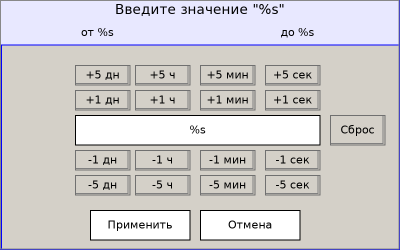
VISUALIZATION TimeInput  // 400x250
VAR_INPUT
	stVariableValue : STRING;
	stMin : STRING;
	stMax : STRING;
	wstTitle : WSTRING;
	flags : DWORD;
END_VAR
VAR
	bInit 			: BOOL;
	stMessage 		: STRING;
	stOutputValue 	: STRING;
	iCaretPosition	: INT;
	iSelectionStart	: INT;
	iSelectionEnd	: INT;
	xAllSelected	: BOOL;
END_VAR
    Rectangle (0,0 400x250)
    Rectangle (200,210 100x30), "Отмена"
        OnMouseDown: CloseDialog Dialog=TimeInput, Result=Cancel, NumpadKeypadSet=True
    Rectangle (90,210 100x30), "Применить"
        OnMouseUp: CloseDialog Dialog=TimeInput, Result=Yes, NumpadKeypad=True, NumpadKeypadSet=True
    Rectangle (0,0 400x45), "Введите значение "%s"", text variable: Header
    Button (265,90 55x20), "+1 сек", invisible if: (MinTime + T#1s >= MaxTime)
        OnMouseUp: execute {
            IF ((timevar+T#1S <= MaxTime ) AND
            			(timevar+T#1S > TimeVar)) THEN
            	timevar:=timevar+T#1S;
            END_IF
        }
    Rectangle (75,115 245x30), "%s", text variable: TIME_TO_WSTRING_HMI(TimeVar)
        p4168582468: "Время"
    Button (265,65 55x20), "+5 сек", invisible if: (MinTime + T#5s >= MaxTime)
        OnMouseUp: execute {
            IF ((timevar+T#5S <= MaxTime ) AND
            			(timevar+T#5S > TimeVar)) THEN
            	timevar:=timevar+T#5S;
            ELSE
            	timevar:=MaxTime;
            END_IF
        }
    Button (265,175 55x20), "-5 сек", invisible if: (MinTime + T#5s) >= MaxTime
        OnMouseUp: execute {
            IF (((timevar-T#5S) >= MinTime)AND
            				(timevar-T#5S < timevar)) THEN
            	timevar:=timevar-T#5S;
            ELSE
            	TimeVar:=MinTime;
            END_IF
        }
    Button (265,150 55x20), "-1 сек", invisible if: (MinTime + T#1s) >= MaxTime
        OnMouseUp: execute {
            IF (((timevar-T#1S) >= MinTime)AND
            				(timevar-T#1S < timevar)) THEN
            	timevar:=timevar-T#1S;
            END_IF
        }
    Button (200,90 55x20), "+1 мин", invisible if: (MinTime + T#1m >= MaxTime)
        OnMouseUp: execute {
            IF ((timevar+T#1M <= MaxTime ) AND
            			(timevar+T#1M > TimeVar)) THEN
            	timevar:=timevar+T#1m;
            END_IF
        }
    Button (200,65 55x20), "+5 мин", invisible if: (MinTime + T#5m > MaxTime)
        OnMouseUp: execute {
            IF ((timevar+T#5M <= MaxTime ) AND
            			(timevar+T#5M > TimeVar)) THEN
            	timevar:=timevar+T#5M;
            ELSE
            	timevar:=MaxTime;
            END_IF
        }
    Button (135,90 55x20), "+1 ч", invisible if: (MinTime + T#1h >= MaxTime)
        OnMouseUp: execute {
            IF ((timevar+T#1H <= MaxTime ) AND
            			(timevar+T#1H > TimeVar)) THEN
            	timevar:=timevar+T#1H;
            END_IF
        }
    Button (135,65 55x20), "+5 ч", invisible if: (MinTime + T#5h >= MaxTime)
        OnMouseUp: execute {
            IF ((timevar+T#5H <= MaxTime ) AND
            			(timevar+T#5H > TimeVar)) THEN
            	timevar:=timevar+T#5h;
            ELSE
            	timevar:=MaxTime;
            END_IF
        }
    Button (200,175 55x20), "-5 мин", invisible if: (MinTime + T#5m) >= MaxTime
        OnMouseUp: execute {
            IF (((timevar-T#5M) >= MinTime)AND
            				(timevar-T#5M < timevar)) THEN
            	timevar:=timevar-T#5m;
            ELSE
            	TimeVar:=MinTime;
            END_IF
        }
    Button (200,150 55x20), "-1 мин", invisible if: (MinTime + T#1m) >=MaxTime
        OnMouseUp: execute {
            IF (((timevar-T#1M) >= MinTime)AND
            				(timevar-T#1M < timevar)) THEN
            	timevar:=timevar-T#1m;
            END_IF
        }
    Button (135,175 55x20), "-5 ч", invisible if: (MinTime + T#5h) >= MaxTime
        OnMouseUp: execute {
            IF (((timevar-T#5H) >= MinTime)AND
            				(timevar-T#5h < timevar)) THEN
            	timevar:=timevar-T#5H;
            ELSE
            	TimeVar:=MinTime;
            END_IF
        }
    Button (135,150 55x20), "-1 ч", invisible if: (MinTime + T#1h) >= MaxTime
        OnMouseUp: execute {
            IF (((timevar-T#1H) >= MinTime)AND
            				(timevar-T#1H < timevar)) THEN
            	timevar:=timevar-T#1h;
            END_IF
        }
    Button (75,90 55x20), "+1 дн", invisible if: (MinTime + T#1d >=MaxTime)
        OnMouseUp: execute {
            IF ((timevar+T#1D <= MaxTime ) AND
            			(timevar+T#1D > TimeVar)) THEN
            	timevar:=timevar+T#1d;
            END_IF
        }
    Button (75,65 55x20), "+5 дн", invisible if: (MinTime + T#5d >= MaxTime)
        OnMouseUp: execute {
            IF ((timevar+T#5D <= MaxTime ) AND
            			(timevar+T#5D > TimeVar)) THEN
            	timevar:=timevar+T#5D;
            ELSE
            	timevar:=MaxTime;
            END_IF
        }
    Button (75,175 55x20), "-5 дн", invisible if: (MinTime + T#5d) >= MaxTime
        OnMouseUp: execute {
            IF (((timevar-T#5D) >= MinTime)AND
            				(timevar-T#5D < timevar)) THEN
            	timevar:=timevar-T#5D;
            ELSE
            	TimeVar:=MinTime;
            END_IF
        }
    Button (75,150 55x20), "-1 дн", invisible if: (MinTime + T#1d) >= MaxTime
        OnMouseUp: execute {
            IF (((timevar-T#1D) >= MinTime)AND
            				(timevar-T#1D < timevar)) THEN
            	timevar:=timevar-T#1D;
            END_IF
        }
    Button (330,115 55x30), "Сброс"
        OnMouseUp: execute { timevar:=MinTime; }
    Rectangle (0,20 195x25), "от %s", text variable: TIME_TO_WSTRING_HMI(MinTime)
        p4168582468: "Время"
    Rectangle (195,20 205x25), "до %s", text variable: TIME_TO_WSTRING_HMI(MaxTime)
        p4168582468: "Время"
    hotkey HotkeyInput Id=481037385728, Key=KeyDown=True, KeyName=ESCAPE, VisuElemId=10
END_VISUALIZATION

(* stored: Version 1.1.0.1, ProductVersion 3.1.4024.4
   Visu TimeInput: Id {0be2a367-d3c2-4cd8-8347-ddd700e41329} *)
